% RSLogix 500 project PLC Level 2 Project 10.RSS, saved by version 8.30.00.16 %
PROJECT "UNTITLED"    % processor: Bul.1763 MicroLogix 1100 Series B %

PROGRAM FILES
  LAD 2 "MAIN"  4 rungs
  LAD 3 "IO CONFIG"  8 rungs
  LAD 4 "CONTROLS"  7 rungs
  LAD 5 "ALARMS"  8 rungs

DATA FILES
  O0 OUTPUT  4 elements
  I1 INPUT  6 elements
  S2 STATUS  66 elements
  B3 BINARY  2 elements
  T4 TIMER  4 elements
  C5 COUNTER  1 elements
  R6 CONTROL  1 elements
  N7 INTEGER  3 elements
  F8 FLOAT  1 elements

LADDER 2 "MAIN"
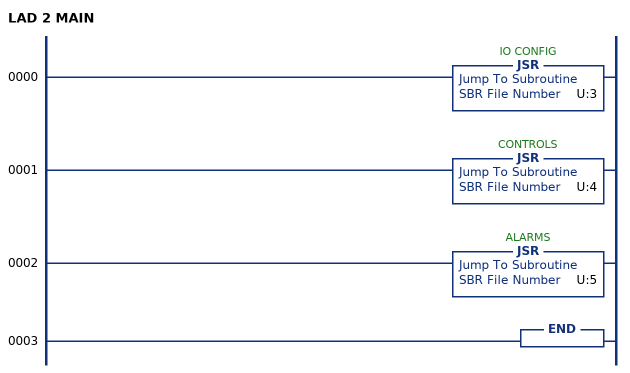
% Rung: 0 %
SOR JSR U:3 EOR
%   U:3  "IO CONFIG" %
% Rung: 1 %
SOR JSR U:4 EOR
%   U:4  "CONTROLS" %
% Rung: 2 %
SOR JSR U:5 EOR
%   U:5  "ALARMS" %
% Rung: 3 %
SOR END EOR

LADDER 3 "IO CONFIG"
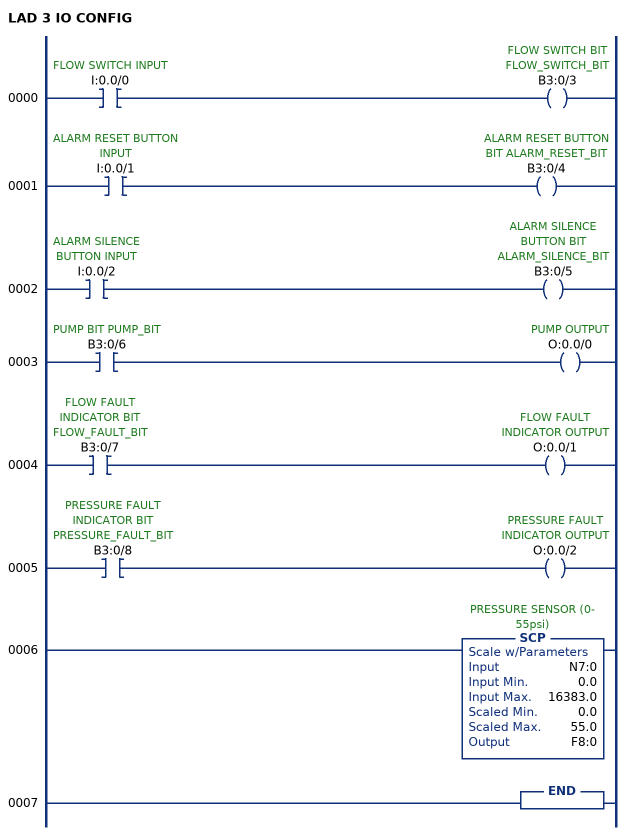
% Rung: 0 %
SOR XIC I:0.0/0 OTE B3:0/3 EOR
%   I:0.0/0  "FLOW SWITCH INPUT" %
%   B3:0/3  FLOW_SWITCH_BIT  "FLOW SWITCH BIT" %
% Rung: 1 %
SOR XIC I:0.0/1 OTE B3:0/4 EOR
%   I:0.0/1  "ALARM RESET BUTTON INPUT" %
%   B3:0/4  ALARM_RESET_BIT  "ALARM RESET BUTTON BIT" %
% Rung: 2 %
SOR XIC I:0.0/2 OTE B3:0/5 EOR
%   I:0.0/2  "ALARM SILENCE BUTTON INPUT" %
%   B3:0/5  ALARM_SILENCE_BIT  "ALARM SILENCE BUTTON BIT" %
% Rung: 3 %
SOR XIC B3:0/6 OTE O:0.0/0 EOR
%   B3:0/6  PUMP_BIT  "PUMP BIT" %
%   O:0.0/0  "PUMP OUTPUT" %
% Rung: 4 %
SOR XIC B3:0/7 OTE O:0.0/1 EOR
%   B3:0/7  FLOW_FAULT_BIT  "FLOW FAULT INDICATOR BIT" %
%   O:0.0/1  "FLOW FAULT INDICATOR OUTPUT" %
% Rung: 5 %
SOR XIC B3:0/8 OTE O:0.0/2 EOR
%   B3:0/8  PRESSURE_FAULT_BIT  "PRESSURE FAULT INDICATOR BIT" %
%   O:0.0/2  "PRESSURE FAULT INDICATOR OUTPUT" %
% Rung: 6 %
SOR SCP N7:0 0.0 16383.0 0.0 55.0 F8:0 EOR
%   N7:0  "PRESSURE SENSOR SIGNAL INPUT" %
%   F8:0  "PRESSURE SENSOR (0- 55psi)" %
% Rung: 7 %
SOR END EOR

LADDER 4 "CONTROLS"
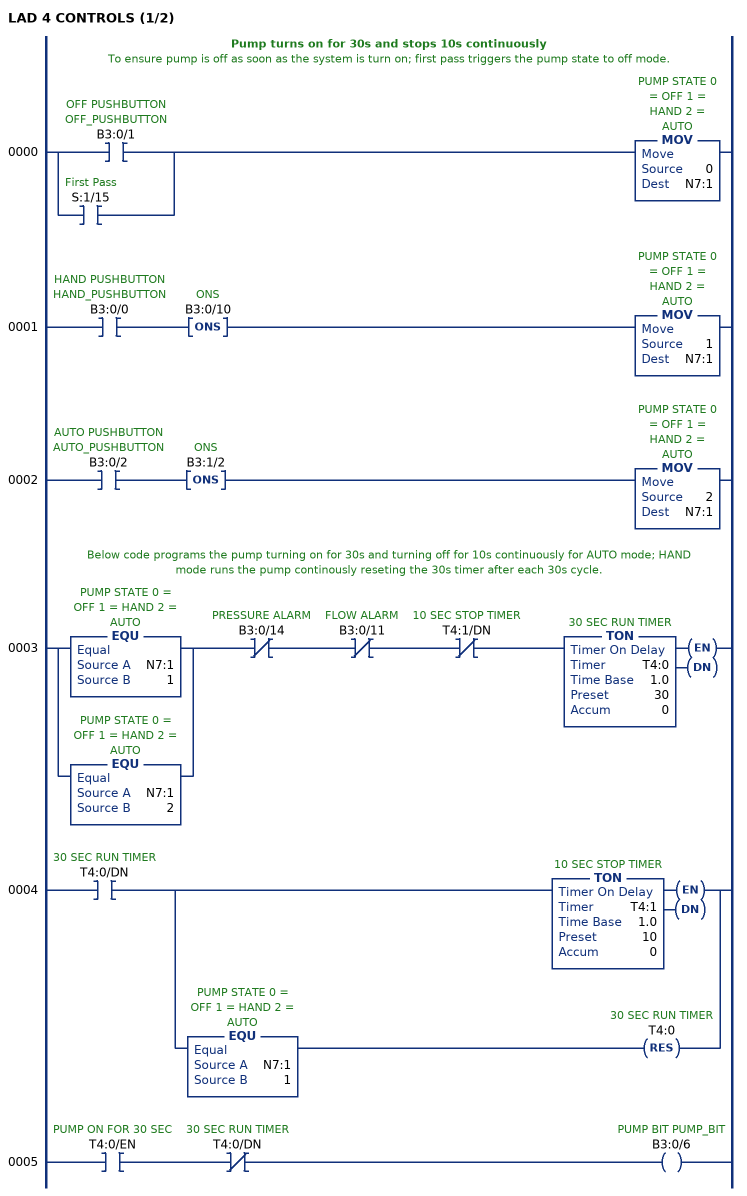
% Rung: 0 %
% TITLE: Pump turns on for 30s and stops 10s continuously %
% To ensure pump is off as soon as the system is turn on; first pass triggers the pump state to off mode. %
SOR BST XIC B3:0/1 NXB XIC S:1/15 BND MOV 0 N7:1 EOR
%   B3:0/1  OFF_PUSHBUTTON  "OFF PUSHBUTTON" %
%   S:1/15  "First Pass" %
%   N7:1  "PUMP STATE 0 = OFF 1 = HAND 2 = AUTO" %
% Rung: 1 %
SOR XIC B3:0/0 ONS B3:0/10 MOV 1 N7:1 EOR
%   B3:0/0  HAND_PUSHBUTTON  "HAND PUSHBUTTON" %
%   B3:0/10  "ONS" %
%   N7:1  "PUMP STATE 0 = OFF 1 = HAND 2 = AUTO" %
% Rung: 2 %
SOR XIC B3:0/2 ONS B3:1/2 MOV 2 N7:1 EOR
%   B3:0/2  AUTO_PUSHBUTTON  "AUTO PUSHBUTTON" %
%   B3:1/2  "ONS" %
%   N7:1  "PUMP STATE 0 = OFF 1 = HAND 2 = AUTO" %
% Rung: 3 %
% Below code programs the pump turning on for 30s and turning off for 10s continuously for AUTO mode; HAND mode runs the pump continously reseting the 30s timer after each 30s cycle. %
SOR BST EQU N7:1 1 NXB EQU N7:1 2 BND XIO B3:0/14 XIO B3:0/11 XIO T4:1/DN TON T4:0 1.0 30 0 EOR
%   N7:1  "PUMP STATE 0 = OFF 1 = HAND 2 = AUTO" %
%   B3:0/14  "PRESSURE ALARM" %
%   B3:0/11  "FLOW ALARM" %
%   T4:1/DN  "10 SEC STOP TIMER" %
%   T4:0  "30 SEC RUN TIMER" %
% Rung: 4 %
SOR XIC T4:0/DN BST TON T4:1 1.0 10 0 NXB EQU N7:1 1 RES T4:0 BND EOR
%   T4:0/DN  "30 SEC RUN TIMER" %
%   T4:1  "10 SEC STOP TIMER" %
%   N7:1  "PUMP STATE 0 = OFF 1 = HAND 2 = AUTO" %
%   T4:0  "30 SEC RUN TIMER" %
% Rung: 5 %
SOR XIC T4:0/EN XIO T4:0/DN OTE B3:0/6 EOR
%   T4:0/EN  "PUMP ON FOR 30 SEC" %
%   T4:0/DN  "30 SEC RUN TIMER" %
%   B3:0/6  PUMP_BIT  "PUMP BIT" %

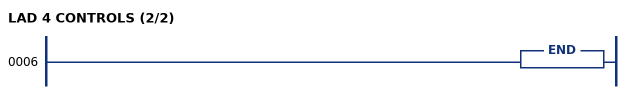
% Rung: 6 %
SOR END EOR

LADDER 5 "ALARMS"
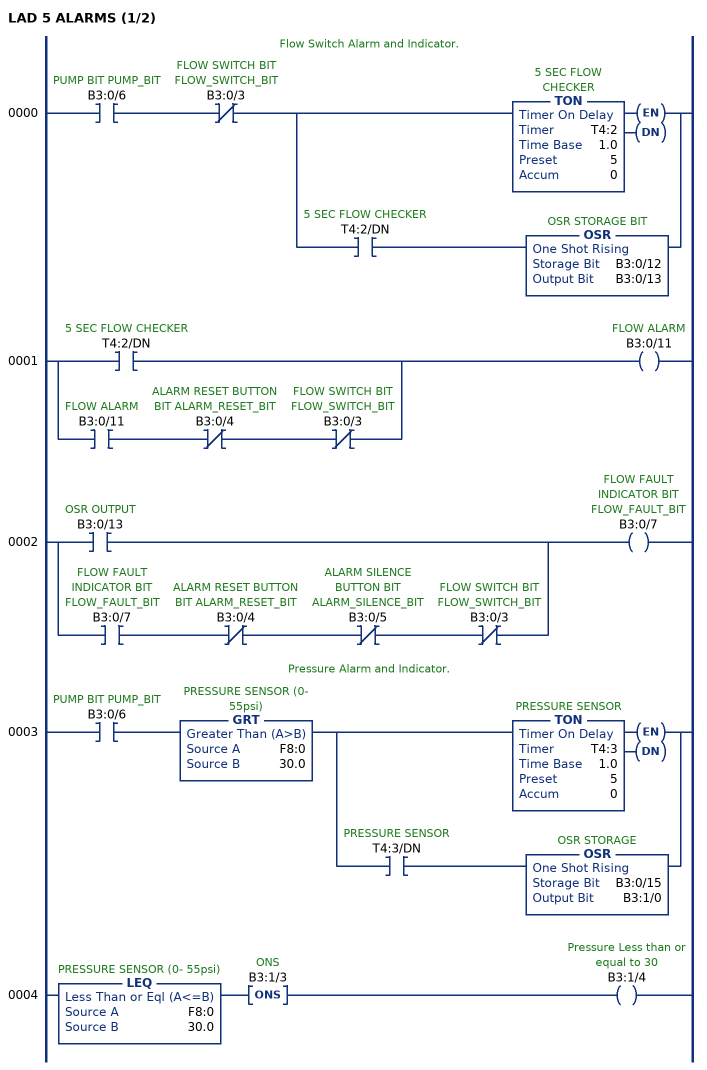
% Rung: 0 %
% Flow Switch Alarm and Indicator. %
SOR XIC B3:0/6 XIO B3:0/3 BST TON T4:2 1.0 5 0 NXB XIC T4:2/DN OSR B3:0/12 B3:0/13 BND EOR
%   B3:0/6  PUMP_BIT  "PUMP BIT" %
%   B3:0/3  FLOW_SWITCH_BIT  "FLOW SWITCH BIT" %
%   T4:2  "5 SEC FLOW CHECKER" %
%   B3:0/12  "OSR STORAGE BIT" %
%   B3:0/13  "OSR OUTPUT" %
% Rung: 1 %
SOR BST XIC T4:2/DN NXB XIC B3:0/11 XIO B3:0/4 XIO B3:0/3 BND OTE B3:0/11 EOR
%   T4:2  "5 SEC FLOW CHECKER" %
%   B3:0/11  "FLOW ALARM" %
%   B3:0/4  ALARM_RESET_BIT  "ALARM RESET BUTTON BIT" %
%   B3:0/3  FLOW_SWITCH_BIT  "FLOW SWITCH BIT" %
% Rung: 2 %
SOR BST XIC B3:0/13 NXB XIC B3:0/7 XIO B3:0/4 XIO B3:0/5 XIO B3:0/3 BND OTE B3:0/7 EOR
%   B3:0/13  "OSR OUTPUT" %
%   B3:0/7  FLOW_FAULT_BIT  "FLOW FAULT INDICATOR BIT" %
%   B3:0/4  ALARM_RESET_BIT  "ALARM RESET BUTTON BIT" %
%   B3:0/5  ALARM_SILENCE_BIT  "ALARM SILENCE BUTTON BIT" %
%   B3:0/3  FLOW_SWITCH_BIT  "FLOW SWITCH BIT" %
% Rung: 3 %
% Pressure Alarm and Indicator. %
SOR XIC B3:0/6 GRT F8:0 30.0 BST TON T4:3 1.0 5 0 NXB XIC T4:3/DN OSR B3:0/15 B3:1/0 BND EOR
%   B3:0/6  PUMP_BIT  "PUMP BIT" %
%   F8:0  "PRESSURE SENSOR (0- 55psi)" %
%   T4:3  "PRESSURE SENSOR" %
%   B3:0/15  "OSR STORAGE" %
%   B3:1/0  "OSR OUTPUT" %
% Rung: 4 %
SOR LEQ F8:0 30.0 ONS B3:1/3 OTE B3:1/4 EOR
%   F8:0  "PRESSURE SENSOR (0- 55psi)" %
%   B3:1/3  "ONS" %
%   B3:1/4  "Pressure Less than or equal to 30" %

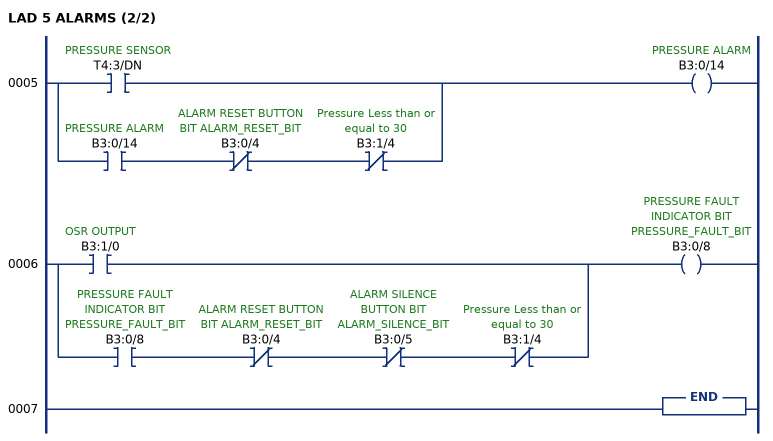
% Rung: 5 %
SOR BST XIC T4:3/DN NXB XIC B3:0/14 XIO B3:0/4 XIO B3:1/4 BND OTE B3:0/14 EOR
%   T4:3  "PRESSURE SENSOR" %
%   B3:0/14  "PRESSURE ALARM" %
%   B3:0/4  ALARM_RESET_BIT  "ALARM RESET BUTTON BIT" %
%   B3:1/4  "Pressure Less than or equal to 30" %
% Rung: 6 %
SOR BST XIC B3:1/0 NXB XIC B3:0/8 XIO B3:0/4 XIO B3:0/5 XIO B3:1/4 BND OTE B3:0/8 EOR
%   B3:1/0  "OSR OUTPUT" %
%   B3:0/8  PRESSURE_FAULT_BIT  "PRESSURE FAULT INDICATOR BIT" %
%   B3:0/4  ALARM_RESET_BIT  "ALARM RESET BUTTON BIT" %
%   B3:0/5  ALARM_SILENCE_BIT  "ALARM SILENCE BUTTON BIT" %
%   B3:1/4  "Pressure Less than or equal to 30" %
% Rung: 7 %
SOR END EOR

OTHER DOCUMENTED ADDRESSES
  B3:0/9  "ONS"
  B3:1/12  "ONS"
  B3:1/13  "ONS"
  B3:1/14  "PUMP TRIGGER"
  N7:2  "PRESSURE SENSOR (0- 55 PSI)"

DATA TABLE (non-zero values as saved)
DATA T4
% .PRE .ACC %
% T4:0 % 30 0
% T4:1 % 10 0
% T4:2 % 5 0
% T4:3 % 5 0
